Staubli VAL3: external.pgx

public program external()
begin
  call external:start()
end
